// TIA Portal project "PICK&PLACE" (V14)

(* hardware
DEVICE "S71500/ET200MP-Station_1"  S7-1500 station
   slot 0: "Profilschiene_0"  6ES7 590-1***0-0AA0
   slot 1: "PLC_1"  CPU 1511-1 PN  6ES7 511-1AK00-0AB0  V1.8
   slot 2: "AI 8xU/I/RTD/TC ST_1"  AI 8xU/I/RTD/TC ST  6ES7 531-7KF00-0AB0  V2.0
   slot 3: "AI 8xU/I/RTD/TC ST_2"  AI 8xU/I/RTD/TC ST  6ES7 531-7KF00-0AB0  V2.0
   slot 4: "AI 8xU/I/RTD/TC ST_3"  AI 8xU/I/RTD/TC ST  6ES7 531-7KF00-0AB0  V2.0
   slot 5: "AI 8xU/I/RTD/TC ST_4"  AI 8xU/I/RTD/TC ST  6ES7 531-7KF00-0AB0  V2.0
   slot 6: "DI 16x24VDC BA_1"  DI 16x24VDC BA  6ES7 521-1BH10-0AA0  V1.0
*)

// ===== PLC "PLC_1"  CPU 1511-1 PN =====

VAR_GLOBAL   // PLC tag table "Standard-Variablentabelle"
   "ON" AT %I1.0 : Bool;
   "Start" AT %I0.4 : Bool;
   "Start Light" AT %Q1.0 : Bool;
   "Stop Light" AT %Q1.2 : Bool;
   "Box conveyor" AT %Q0.0 : Bool;
   "Part at place" AT %I0.1 : Bool;
   "Part conveyor" AT %Q0.1 : Bool;
   "Tag_1" AT %M0.6 : Bool;
   "Tag_2" AT %M0.0 : Bool;
   "SPX" AT %QD30 : Real;
   "SPY" AT %QD34 : Real;
   "Box at place" AT %I0.0 : Bool;
   "Tag_3" AT %M1.1 : Bool;
   "X" AT %ID30 : DWord;
   "Grab" AT %Q0.4 : Bool;
   "Y" AT %ID34 : Real;
   "SPZ" AT %QD38 : Real;
   "Detected" AT %I0.2 : Bool;
   "Tag_4" AT %M0.1 : Bool;
   "Tag_5" AT %M0.4 : Bool;
   "Z" AT %ID38 : Real;
   "Tag_7" AT %M0.2 : Bool;
   "Tag_8" AT %M0.3 : Bool;
   "Tag_9" AT %M0.5 : Bool;
   "C+" AT %Q0.3 : Bool;
   "Exit conveyor" AT %Q0.2 : Bool;
   "Exit Green" AT %Q0.5 : Bool;
   "Tag_6" AT %M1.0 : Bool;
   "Tag_10" AT %MB0 : Byte;
   "Counter" AT %QD42 : DInt;
   "Reset" AT %I0.5 : Bool;
   "Reset Light" AT %Q1.1 : Bool;
   "Stop" AT %I0.6 : Bool;
   "Tag_11" AT %QB0 : Byte;
   "Tag_12" AT %MB1 : Byte;
   "OFF" AT %I1.1 : Bool;
   "BCstart" AT %I1.3 : Bool;
   "BCstop" AT %I1.4 : Bool;
   "ECstart" AT %I1.6 : Bool;
   "ECstop" AT %I1.7 : Bool;
END_VAR

// folder: System blocks/Program resources

DATA_BLOCK "IEC_Timer_0_DB"   // DB1
{ S7_Optimized_Access := 'TRUE' }
AUTHOR : Simatic
FAMILY : IEC
NAME : IEC_TMR
VERSION : 1.0
// stored: InstanceOfName IEC_TIMER
"IEC_TIMER"
BEGIN
END_DATA_BLOCK

DATA_BLOCK "IEC_Timer_0_DB_1"   // DB2
{ S7_Optimized_Access := 'TRUE' }
AUTHOR : Simatic
FAMILY : IEC
NAME : IEC_TMR
VERSION : 1.0
// stored: InstanceOfName IEC_TIMER
"IEC_TIMER"
BEGIN
END_DATA_BLOCK

DATA_BLOCK "IEC_Timer_0_DB_2"   // DB3
{ S7_Optimized_Access := 'TRUE' }
AUTHOR : Simatic
FAMILY : IEC
NAME : IEC_TMR
VERSION : 1.0
// stored: InstanceOfName IEC_TIMER
"IEC_TIMER"
BEGIN
END_DATA_BLOCK

DATA_BLOCK "IEC_Timer_0_DB_3"   // DB4
{ S7_Optimized_Access := 'TRUE' }
AUTHOR : Simatic
FAMILY : IEC
NAME : IEC_TMR
VERSION : 1.0
// stored: InstanceOfName IEC_TIMER
"IEC_TIMER"
BEGIN
END_DATA_BLOCK

DATA_BLOCK "IEC_Timer_0_DB_4"   // DB5
{ S7_Optimized_Access := 'TRUE' }
AUTHOR : Simatic
FAMILY : IEC
NAME : IEC_TMR
VERSION : 1.0
// stored: InstanceOfName IEC_TIMER
"IEC_TIMER"
BEGIN
END_DATA_BLOCK

DATA_BLOCK "IEC_Timer_0_DB_5"   // DB6
{ S7_Optimized_Access := 'TRUE' }
AUTHOR : Simatic
FAMILY : IEC
NAME : IEC_TMR
VERSION : 1.0
// stored: InstanceOfName IEC_TIMER
"IEC_TIMER"
BEGIN
END_DATA_BLOCK

DATA_BLOCK "IEC_Timer_0_DB_6"   // DB7
{ S7_Optimized_Access := 'TRUE' }
AUTHOR : Simatic
FAMILY : IEC
NAME : IEC_TMR
VERSION : 1.0
// stored: InstanceOfName IEC_TIMER
"IEC_TIMER"
BEGIN
END_DATA_BLOCK

// folder: (top level)

FUNCTION "MHJ-PLC-Lab-Function-S71500" : Void   // FC9000, SCL
{ S7_Optimized_Access := 'TRUE' }
VERSION : 0.1
   VAR_TEMP
      Value : Byte;
      ForCounter : Int;
   END_VAR
   VAR CONSTANT
      Value_01_DW : DWord := 16#1223_5486;
      Value_02_DW : DWord := 16#A6C9_D1F5;
   END_VAR
BEGIN

   #Value:=PEEK(area := 16#82,
        dbNumber := 0,
        byteOffset := 511);
   #Value := #Value + 1;

   POKE(area := 16#82,
        dbNumber := 0,
        byteOffset := 511,
        value := #Value);

   POKE(area := 16#82,
        dbNumber := 0,
        byteOffset := 1016,
        value := #Value_01_DW);
   POKE(area := 16#82,
        dbNumber := 0,
        byteOffset := 1020,
        value := #Value_02_DW);

   FOR #ForCounter := 0 TO 63 DO
       #Value:=PEEK(area := 16#1,
            dbNumber := 0,
            byteOffset := #ForCounter);
       POKE(area := 16#81,
            dbNumber := 0,
            byteOffset := #ForCounter,
            value := #Value);
   END_FOR;
   #Value := PEEK(area := 16#1,
                  dbNumber := 0,
                  byteOffset := 512);
   POKE(area := 16#82,
        dbNumber := 0,
        byteOffset := 512,
        value := #Value);
END_FUNCTION

ORGANIZATION_BLOCK "Main"   // OB1, LAD, ProgramCycle
TITLE = "Main Program Sweep (Cycle)"
{ S7_Optimized_Access := 'TRUE' }
VERSION : 0.1
   VAR_INPUT
      Initial_Call : Bool;   // Initial call of this OB
      Remanence : Bool;   // =True, if remanent data are available
   END_VAR
   VAR_TEMP   // added for the SCL form of the ladder/FBD networks
      _w1 : Bool;
      _w2 : Bool;
      _w3 : Bool;
      _w4 : Bool;
      _w5 : Bool;
      _w6 : Bool;
      _w7 : Bool;
      _w8 : Bool;
      _w9 : Bool;
      _w10 : Bool;
      _w11 : Bool;
      _w12 : Bool;
      _w13 : Bool;
   END_VAR
BEGIN

REGION Network 1
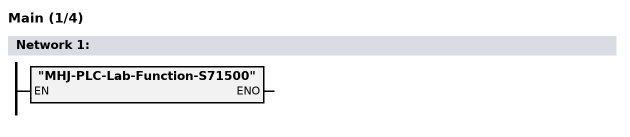
   RUNG wire#powerrail
      "MHJ-PLC-Lab-Function-S71500"()
   END_RUNG
   // the same network as SCL:
   "MHJ-PLC-Lab-Function-S71500"();
END_REGION

REGION Network 2
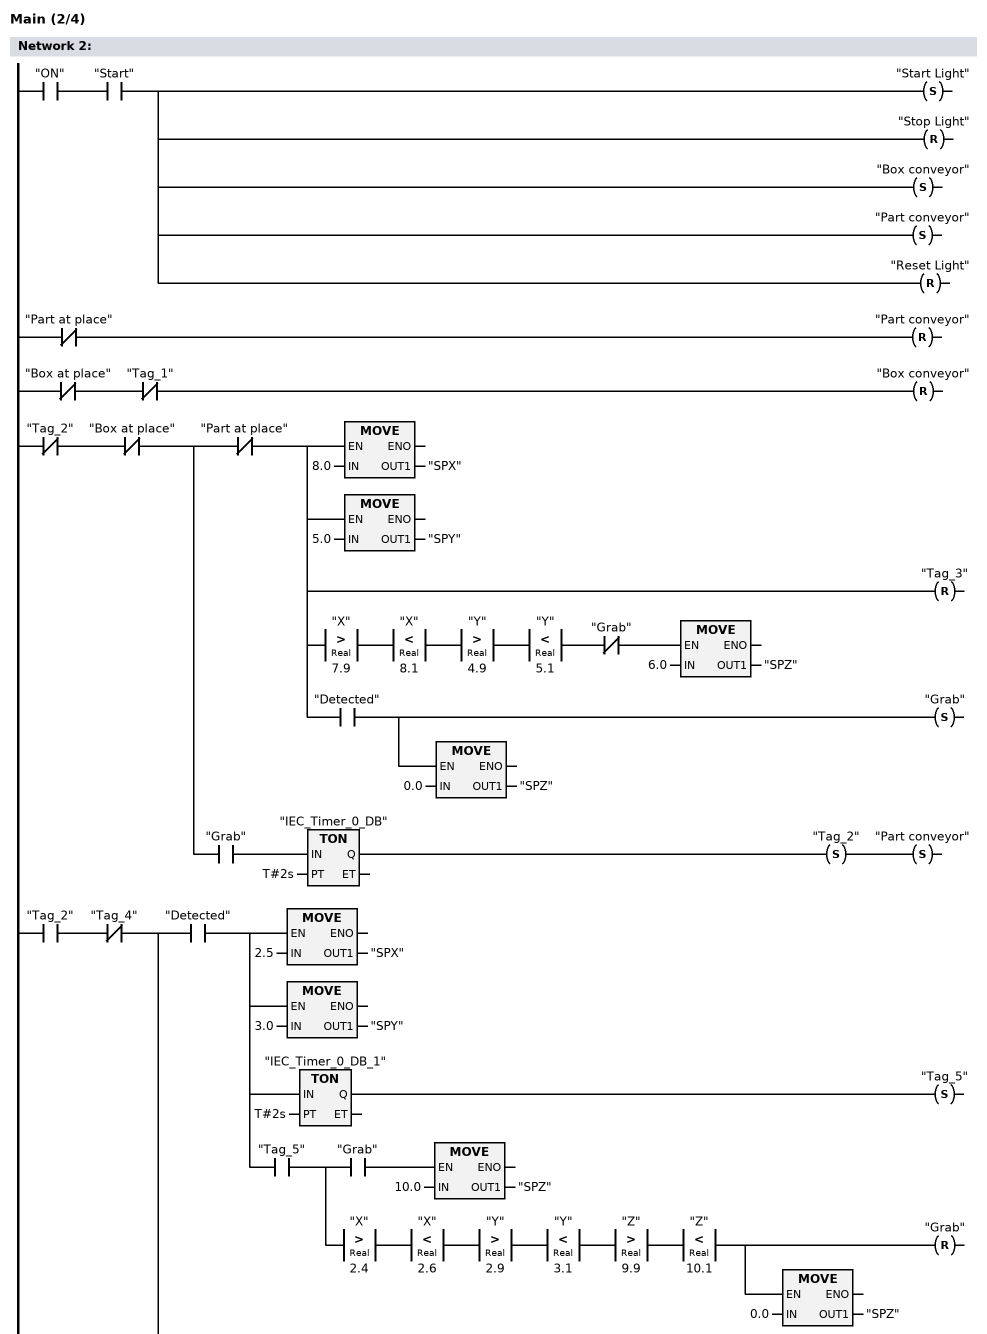
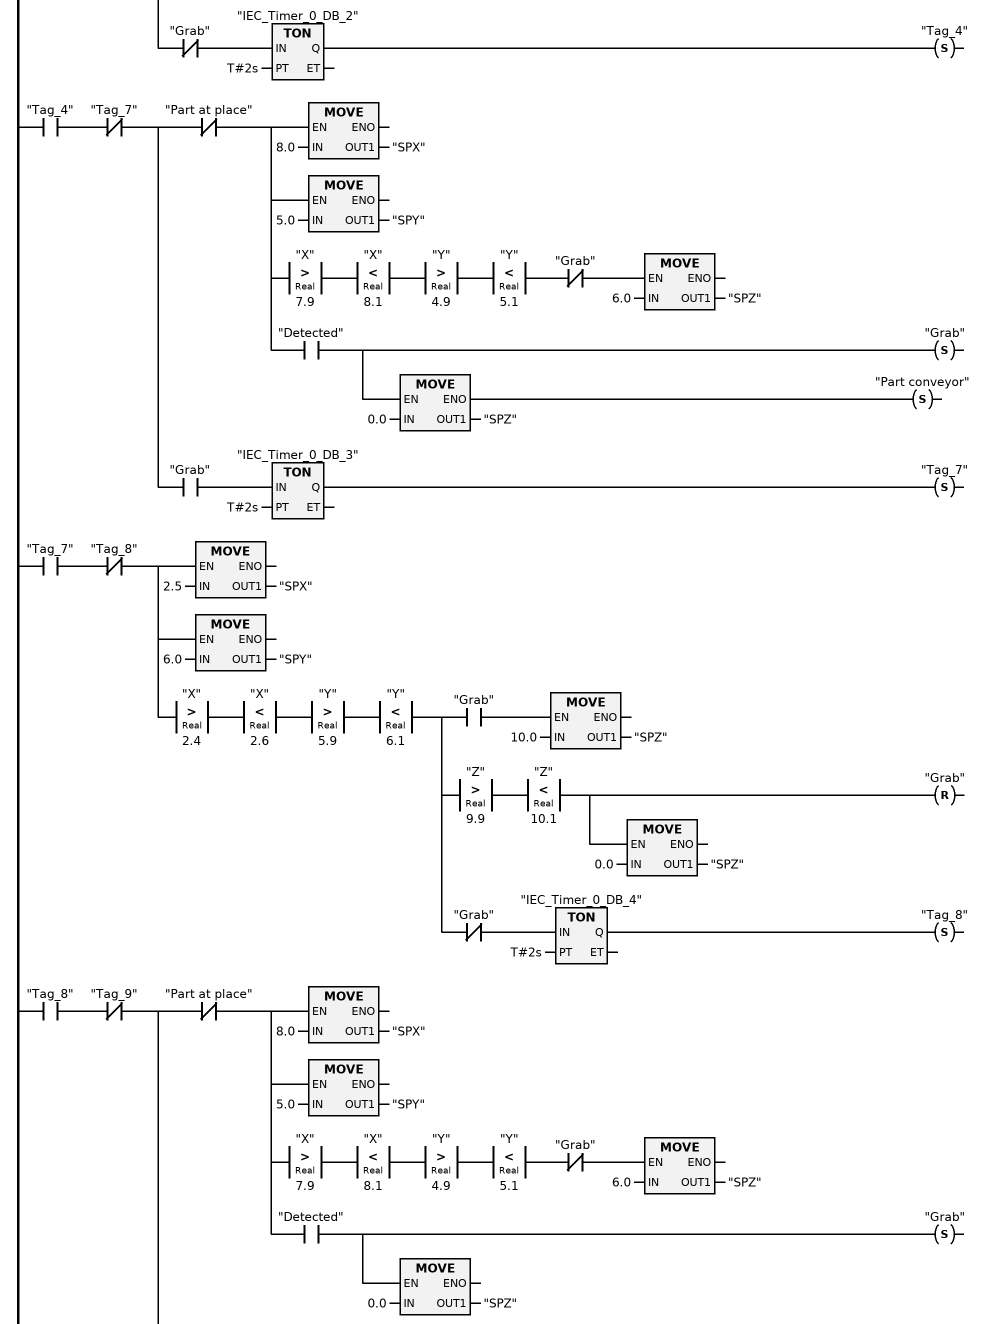
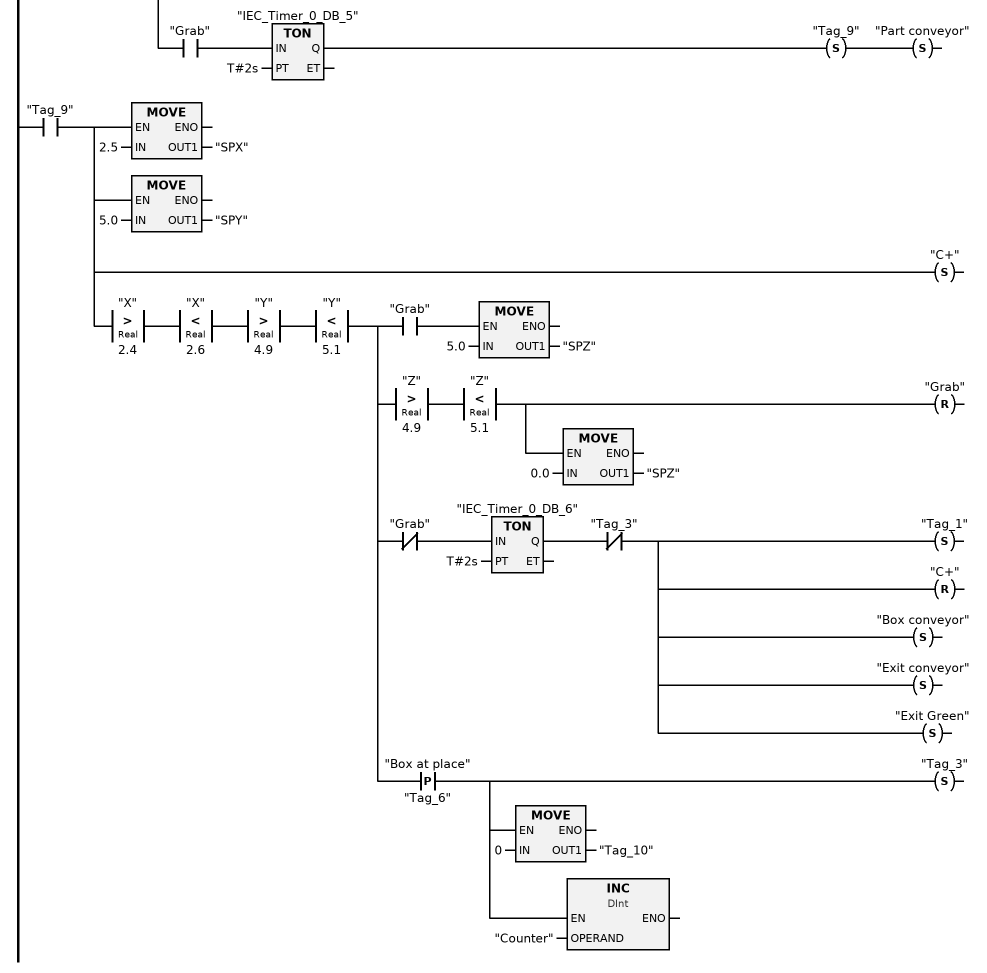
   IF "ON" AND "Start" THEN
       "Start Light" := TRUE;
       "Stop Light" := FALSE;
       "Box conveyor" := TRUE;
       "Part conveyor" := TRUE;
       "Reset Light" := FALSE;
   END_IF;
   IF NOT "Part at place" THEN "Part conveyor" := FALSE; END_IF;
   IF NOT "Box at place" AND NOT "Tag_1" THEN "Box conveyor" := FALSE; END_IF;
   #_w1 := NOT "Tag_2" AND NOT "Box at place";
   #_w2 := #_w1 AND NOT "Part at place";
   IF #_w2 THEN
       "SPX" := 8.0;
       "SPY" := 5.0;
       "Tag_3" := FALSE;
   END_IF;
   IF #_w2 AND ("X" > 7.9) AND ("X" < 8.1) AND ("Y" > 4.9) AND ("Y" < 5.1) AND NOT "Grab" THEN
       "SPZ" := 6.0;
   END_IF;
   IF #_w2 AND "Detected" THEN
       "Grab" := TRUE;
       "SPZ" := 0.0;
   END_IF;
   "IEC_Timer_0_DB".TON(IN := #_w1 AND "Grab", PT := T#2s);
   IF "IEC_Timer_0_DB".Q THEN
       "Tag_2" := TRUE;
       "Part conveyor" := TRUE;
   END_IF;
   #_w3 := "Tag_2" AND NOT "Tag_4";
   #_w4 := #_w3 AND "Detected";
   IF #_w4 THEN
       "SPX" := 2.5;
       "SPY" := 3.0;
   END_IF;
   "IEC_Timer_0_DB_1".TON(IN := #_w4, PT := T#2s);
   IF "IEC_Timer_0_DB_1".Q THEN "Tag_5" := TRUE; END_IF;
   #_w5 := #_w4 AND "Tag_5";
   IF #_w5 AND "Grab" THEN "SPZ" := 10.0; END_IF;
   IF #_w5 AND ("X" > 2.4) AND ("X" < 2.6) AND ("Y" > 2.9) AND ("Y" < 3.1) AND ("Z" > 9.9) AND ("Z" < 10.1) THEN
       "Grab" := FALSE;
       "SPZ" := 0.0;
   END_IF;
   "IEC_Timer_0_DB_2".TON(IN := #_w3 AND NOT "Grab", PT := T#2s);
   IF "IEC_Timer_0_DB_2".Q THEN "Tag_4" := TRUE; END_IF;
   #_w6 := "Tag_4" AND NOT "Tag_7";
   #_w7 := #_w6 AND NOT "Part at place";
   IF #_w7 THEN
       "SPX" := 8.0;
       "SPY" := 5.0;
   END_IF;
   IF #_w7 AND ("X" > 7.9) AND ("X" < 8.1) AND ("Y" > 4.9) AND ("Y" < 5.1) AND NOT "Grab" THEN
       "SPZ" := 6.0;
   END_IF;
   IF #_w7 AND "Detected" THEN
       "Grab" := TRUE;
       "SPZ" := 0.0;
       "Part conveyor" := TRUE;
   END_IF;
   "IEC_Timer_0_DB_3".TON(IN := #_w6 AND "Grab", PT := T#2s);
   IF "IEC_Timer_0_DB_3".Q THEN "Tag_7" := TRUE; END_IF;
   #_w8 := "Tag_7" AND NOT "Tag_8";
   IF #_w8 THEN
       "SPX" := 2.5;
       "SPY" := 6.0;
   END_IF;
   #_w9 := #_w8 AND ("X" > 2.4) AND ("X" < 2.6) AND ("Y" > 5.9) AND ("Y" < 6.1);
   IF #_w9 AND "Grab" THEN "SPZ" := 10.0; END_IF;
   IF #_w9 AND ("Z" > 9.9) AND ("Z" < 10.1) THEN
       "Grab" := FALSE;
       "SPZ" := 0.0;
   END_IF;
   "IEC_Timer_0_DB_4".TON(IN := #_w9 AND NOT "Grab", PT := T#2s);
   IF "IEC_Timer_0_DB_4".Q THEN "Tag_8" := TRUE; END_IF;
   #_w10 := "Tag_8" AND NOT "Tag_9";
   #_w11 := #_w10 AND NOT "Part at place";
   IF #_w11 THEN
       "SPX" := 8.0;
       "SPY" := 5.0;
   END_IF;
   IF #_w11 AND ("X" > 7.9) AND ("X" < 8.1) AND ("Y" > 4.9) AND ("Y" < 5.1) AND NOT "Grab" THEN
       "SPZ" := 6.0;
   END_IF;
   IF #_w11 AND "Detected" THEN
       "Grab" := TRUE;
       "SPZ" := 0.0;
   END_IF;
   "IEC_Timer_0_DB_5".TON(IN := #_w10 AND "Grab", PT := T#2s);
   IF "IEC_Timer_0_DB_5".Q THEN
       "Tag_9" := TRUE;
       "Part conveyor" := TRUE;
   END_IF;
   IF "Tag_9" THEN
       "SPX" := 2.5;
       "SPY" := 5.0;
       "C+" := TRUE;
   END_IF;
   #_w12 := "Tag_9" AND ("X" > 2.4) AND ("X" < 2.6) AND ("Y" > 4.9) AND ("Y" < 5.1);
   IF #_w12 AND "Grab" THEN "SPZ" := 5.0; END_IF;
   IF #_w12 AND ("Z" > 4.9) AND ("Z" < 5.1) THEN
       "Grab" := FALSE;
       "SPZ" := 0.0;
   END_IF;
   "IEC_Timer_0_DB_6".TON(IN := #_w12 AND NOT "Grab", PT := T#2s);
   IF "IEC_Timer_0_DB_6".Q AND NOT "Tag_3" THEN
       "Tag_1" := TRUE;
       "C+" := FALSE;
       "Box conveyor" := TRUE;
       "Exit conveyor" := TRUE;
       "Exit Green" := TRUE;
   END_IF;
   #_w13 := #_w12 AND "Box at place" AND NOT "Tag_6";   // rising edge of "Box at place"
   "Tag_6" := "Box at place";
   IF #_w13 THEN
       "Tag_3" := TRUE;
       "Tag_10" := 0;
       "Counter" := "Counter" + 1;
   END_IF;
END_REGION

REGION Network 3
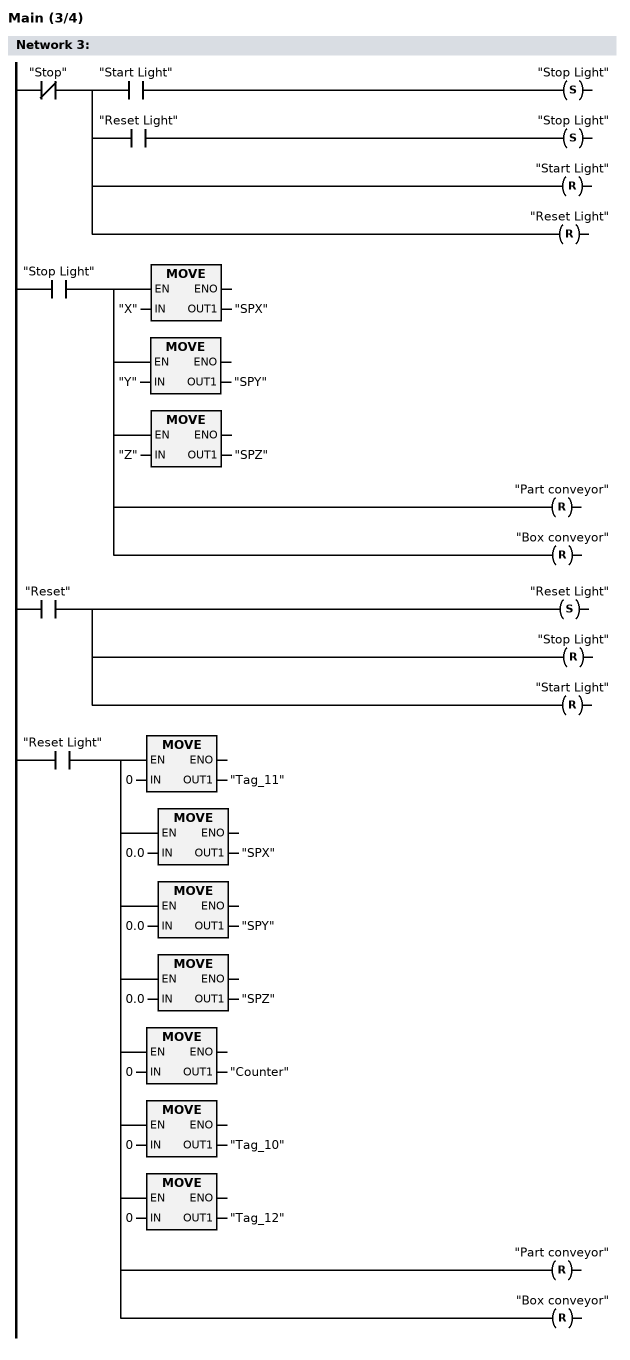
   RUNG wire#powerrail
      I_Contact( "Stop" )
      wire#w1
      Contact( "Start Light" )
      S_Coil( "Stop Light" )
   END_RUNG
   RUNG wire#w1
      Contact( "Reset Light" )
      S_Coil( "Stop Light" )
   END_RUNG
   RUNG wire#w1
      R_Coil( "Start Light" )
   END_RUNG
   RUNG wire#w1
      R_Coil( "Reset Light" )
   END_RUNG
   RUNG wire#powerrail
      Contact( "Stop Light" )
      wire#w2
      Move(in := "X", out1 => "SPX")
   END_RUNG
   RUNG wire#w2
      Move(in := "Y", out1 => "SPY")
   END_RUNG
   RUNG wire#w2
      Move(in := "Z", out1 => "SPZ")
   END_RUNG
   RUNG wire#w2
      R_Coil( "Part conveyor" )
   END_RUNG
   RUNG wire#w2
      R_Coil( "Box conveyor" )
   END_RUNG
   RUNG wire#powerrail
      Contact( "Reset" )
      wire#w3
      S_Coil( "Reset Light" )
   END_RUNG
   RUNG wire#w3
      R_Coil( "Stop Light" )
   END_RUNG
   RUNG wire#w3
      R_Coil( "Start Light" )
   END_RUNG
   RUNG wire#powerrail
      Contact( "Reset Light" )
      wire#w4
      Move(in := 0, out1 => "Tag_11")
   END_RUNG
   RUNG wire#w4
      Move(in := 0.0, out1 => "SPX")
   END_RUNG
   RUNG wire#w4
      Move(in := 0.0, out1 => "SPY")
   END_RUNG
   RUNG wire#w4
      Move(in := 0.0, out1 => "SPZ")
   END_RUNG
   RUNG wire#w4
      Move(in := 0, out1 => "Counter")
   END_RUNG
   RUNG wire#w4
      Move(in := 0, out1 => "Tag_10")
   END_RUNG
   RUNG wire#w4
      Move(in := 0, out1 => "Tag_12")
   END_RUNG
   RUNG wire#w4
      R_Coil( "Part conveyor" )
   END_RUNG
   RUNG wire#w4
      R_Coil( "Box conveyor" )
   END_RUNG
   // the same network as SCL:
   IF NOT "Stop" AND "Start Light" THEN "Stop Light" := TRUE; END_IF;
   IF NOT "Stop" AND "Reset Light" THEN "Stop Light" := TRUE; END_IF;
   IF NOT "Stop" THEN
       "Start Light" := FALSE;
       "Reset Light" := FALSE;
   END_IF;
   IF "Stop Light" THEN
       "SPX" := "X";
       "SPY" := "Y";
       "SPZ" := "Z";
       "Part conveyor" := FALSE;
       "Box conveyor" := FALSE;
   END_IF;
   IF "Reset" THEN
       "Reset Light" := TRUE;
       "Stop Light" := FALSE;
       "Start Light" := FALSE;
   END_IF;
   IF "Reset Light" THEN
       "Tag_11" := 0;
       "SPX" := 0.0;
       "SPY" := 0.0;
       "SPZ" := 0.0;
       "Counter" := 0;
       "Tag_10" := 0;
       "Tag_12" := 0;
       "Part conveyor" := FALSE;
       "Box conveyor" := FALSE;
   END_IF;
END_REGION

REGION Network 4
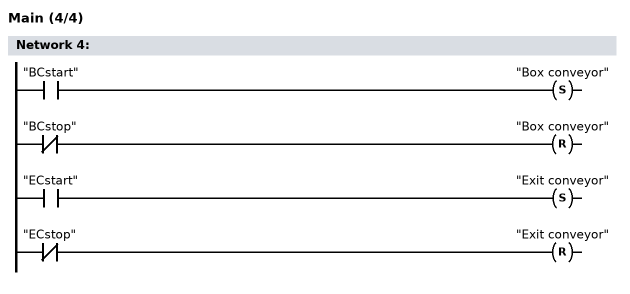
   RUNG wire#powerrail
      Contact( "BCstart" )
      S_Coil( "Box conveyor" )
   END_RUNG
   RUNG wire#powerrail
      I_Contact( "BCstop" )
      R_Coil( "Box conveyor" )
   END_RUNG
   RUNG wire#powerrail
      Contact( "ECstart" )
      S_Coil( "Exit conveyor" )
   END_RUNG
   RUNG wire#powerrail
      I_Contact( "ECstop" )
      R_Coil( "Exit conveyor" )
   END_RUNG
   // the same network as SCL:
   IF "BCstart" THEN "Box conveyor" := TRUE; END_IF;
   IF NOT "BCstop" THEN "Box conveyor" := FALSE; END_IF;
   IF "ECstart" THEN "Exit conveyor" := TRUE; END_IF;
   IF NOT "ECstop" THEN "Exit conveyor" := FALSE; END_IF;
END_REGION
END_ORGANIZATION_BLOCK